// TIA Portal project "lab2" (V15)

(* hardware
DEVICE "S7-1200 station_1"  S7-1200 Station
   slot 0: "Rack_0"  S7-1200 Rack  Rack  V1.0
   slot 1: "PLC_1"  CPU 1214C DC/DC/DC  6ES7 214-1AG40-0XB0  V4.2
      slot 3: "AQ 1x12BIT_1"  AQ1 signal board  6ES7 232-4HA30-0XB0  V1.0
   slot 101: "CM 1243-5"  CM 1243-5  6GK7 243-5DX30-0XE0  V1.3
   slot 102: "CM 1241 (RS485)_1"  CM 1241 (RS485)  6ES7 241-1CH30-0XB0  V1.0
*)

// ===== PLC "PLC_1"  CPU 1214C DC/DC/DC =====

VAR_GLOBAL   // PLC tag table "Default tag table"
   "start" AT %I0.0 : Bool;
   "przerwanie" AT %Q0.0 : Bool;
   "stop" AT %I0.1 : Bool;
   "zaklocenie1" AT %I0.2 : Bool;
   "alarm" AT %Q0.3 : Bool;
   "kasowanie" AT %I0.7 : Bool;
   "przerwanie(1)" AT %Q0.2 : Bool;
   "Tag_2" AT %Q0.5 : Bool;
END_VAR

ORGANIZATION_BLOCK "Main"   // OB1, LAD, ProgramCycle
TITLE = "Main Program Sweep (Cycle)"
{ S7_Optimized_Access := 'TRUE' }
VERSION : 0.1
   VAR_INPUT
      Initial_Call : Bool;   // Initial call of this OB
      Remanence : Bool;   // =True, if remanent data are available
   END_VAR
BEGIN

REGION Network 1: zapis z dominacja kasowania
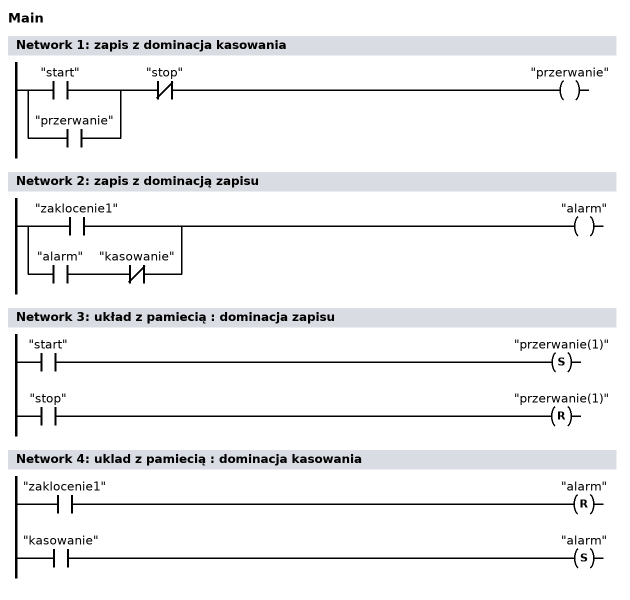
   RUNG wire#powerrail
      Contact( "start" )
      wire#w1
      I_Contact( "stop" )
      Coil( "przerwanie" )
   END_RUNG
   RUNG wire#powerrail
      Contact( "przerwanie" )
   END_RUNG wire#w1
   // the same network as SCL:
   "przerwanie" := ("start" OR "przerwanie") AND NOT "stop";
END_REGION

REGION Network 2: zapis z dominacją zapisu
   RUNG wire#powerrail
      Contact( "zaklocenie1" )
      wire#w1
      Coil( "alarm" )
   END_RUNG
   RUNG wire#powerrail
      Contact( "alarm" )
      I_Contact( "kasowanie" )
   END_RUNG wire#w1
   // the same network as SCL:
   "alarm" := "zaklocenie1" OR ("alarm" AND NOT "kasowanie");
END_REGION

REGION Network 3: układ z pamiecią : dominacja zapisu
   RUNG wire#powerrail
      Contact( "start" )
      S_Coil( "przerwanie(1)" )
   END_RUNG
   RUNG wire#powerrail
      Contact( "stop" )
      R_Coil( "przerwanie(1)" )
   END_RUNG
   // the same network as SCL:
   IF "start" THEN "przerwanie(1)" := TRUE; END_IF;
   IF "stop" THEN "przerwanie(1)" := FALSE; END_IF;
END_REGION

REGION Network 4: uklad z pamiecią : dominacja kasowania
   RUNG wire#powerrail
      Contact( "zaklocenie1" )
      R_Coil( "alarm" )
   END_RUNG
   RUNG wire#powerrail
      Contact( "kasowanie" )
      S_Coil( "alarm" )
   END_RUNG
   // the same network as SCL:
   IF "zaklocenie1" THEN "alarm" := FALSE; END_IF;
   IF "kasowanie" THEN "alarm" := TRUE; END_IF;
END_REGION
END_ORGANIZATION_BLOCK